TYPE Status_ModbusRTU : (Aktiv, ConfigPT, ConfigEV, ConfigMSS);
END_TYPE

(* stored: Version 1.1.0.1, ProductVersion 3.1.4018.5
   DUT Status_ModbusRTU: Id {67b55078-28ad-48b5-ba23-2eb7cd7fc8cc} *)
